
FUNCTION CB_dword_to_real : REAL


TITLE = ' Convert a dword into a real '
VERSION : '1.0'
AUTHOR  : CB
NAME    : dworToRe
FAMILY  : TNI

VAR_INPUT
    IN : DWORD;
END_VAR

BEGIN
CB_dword_to_real := DINT_TO_REAL(DWORD_TO_DINT(IN));

END_FUNCTION
